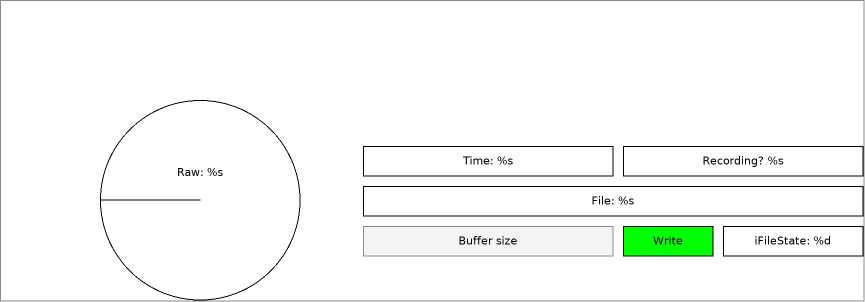
VISUALIZATION Visualization  // 865x302
    Rectangle (623,146 240x30), "Recording? %s", text variable: MAIN.bRecordData
        OnMouseDown: execute { MAIN.bRecordData := NOT MAIN.bRecordData; }
    Ellipse (100,100 200x200), "Raw: %s", text variable: MAIN.enc_raw
    Line (200,200) (100,200)
        p2858320360: MAIN.enc_angle
    Progressbar (363,226 250x30), "Buffer size", variable: MAIN.iEndOfBuffer
    Rectangle (623,226 90x30), "Write", text variable: MAIN.bRecordData, invisible if: not MAIN.fbFileWriter.bBusy
    Rectangle (723,226 140x30), "iFileState: %d", text variable: MAIN.iFileState
    Rectangle (363,146 250x30), "Time: %s", text variable: MAIN.sTime
    Rectangle (363,186 500x30), "File: %s", text variable: MAIN.sFileName
END_VISUALIZATION

(* stored: Version 1.1.0.1, ProductVersion 3.1.4022.10
   Visu Visualization: Id {34b664a4-8d8d-4b1d-a719-b54764bdbfc9} *)
